FUNCTION_BLOCK AOI_StagingTemplate
VAR_INPUT
	execute : BOOL;
END_VAR
VAR_IN_OUT
	materialsArr : ARRAY[*] OF PositionMaterials; //[0..GVL.maxPairs]
	table : StagingTable;
END_VAR
VAR_INPUT
	includeTop, includeLeft, includeRight, includeBottom : BOOL; 
END_VAR
VAR_OUTPUT
	busy : BOOL;
	done : BOOL;
END_VAR
VAR
	trigger : R_TRIG;
	run : BOOL;
	step : (IDLE, GENERATE, COMPLETE);
	i : INT;
END_VAR
VAR	
	stagingArray : ARRAY[0..(GVL.maxPairs+1)*2] OF STRING;
	
	template : StagingTable;
	templateSlots AT %M* : ARRAY[1..10] OF MaterialSlot;
END_VAR

{warning disable C0371}

template(slots:= templateSlots);

trigger(CLK:= execute, Q=> run);

CASE step OF
	IDLE:
		IF run THEN
			step := GENERATE;
			done := FALSE;
		END_IF
		
	GENERATE:
		//strings contain garbage chars after a null byte, they must be manually cleaned before checking if they are byte-empty
		CleanStringsArray(arr := stagingArray);
		IF ArrayIsEmpty(arr := ADR(stagingArray), arrSize := SIZEOF(stagingArray)) THEN //if staging array is empty, fill the array
			createStagingArray(
				includeTop:= includeTop, 
				includeLeft:= includeLeft, 
				includeRight:= includeRight, 
				includeBottom:= includeBottom);
		END_IF
		
		//copy over the real slots before autofilling, otherwise the template may fill occupied slots
		table.copyFrom(src := table);
		
		(*
		iterate through all pairs and autofill the template
		replace succesfully autofilled materials with empty string
		if staging needs to be performed a 2nd time, autofilling empty strings is always unsuccessful
		*)
		FOR i:=0 TO (GVL.maxPairs+1)*2 BY 1 DO
			IF template.autofill(material := stagingArray[i]) THEN
				stagingArray[i] := '';
			END_IF
		END_FOR
		
		step := COMPLETE;
	
	COMPLETE:
		done := TRUE;
		
		step := IDLE;
		
END_CASE

busy := run OR step > 0;

METHOD PRIVATE addToStagingArray : BOOL
VAR_INPUT
	material : STRING;
END_VAR
VAR
	remainingMaterial : STRING;
	splitMaterial : STRING;
END_VAR
remainingMaterial := material;
WHILE FIND(remainingMaterial, '_') > 0 DO
	splitCombinedMaterials(remainingMaterial, splitMaterial);
	IF splitMaterial <> '' THEN
		AddToStringArray(arr := stagingArray, newString := splitMaterial, numElements => , nextIndex => );
		(*
		AddToArray(
			arr := ADR(stagingArray), 
			numEntries := SIZEOF(stagingArray)/SIZEOF(stagingArray[0]), 
			dataSize := SIZEOF(STRING), 
			newEntry := splitMaterial);
		*)
	END_IF
END_WHILE

IF remainingMaterial <> '' THEN
	AddToStringArray(arr := stagingArray, newString := remainingMaterial, numElements => , nextIndex => );
	(*
	AddToArray(
		arr := ADR(stagingArray), 
		numEntries := SIZEOF(stagingArray)/SIZEOF(stagingArray[0]), 
		dataSize := SIZEOF(STRING), 
		newEntry := remainingMaterial);
	*)
END_IF

addToStagingArray := TRUE;
END_METHOD

METHOD clearArray : BOOL
VAR_INPUT
END_VAR
MEMSET(ADR(stagingArray), 0, SIZEOF(stagingArray));
END_METHOD

METHOD clearTemplate : BOOL
VAR_INPUT
END_VAR
template.clear();
END_METHOD

METHOD PRIVATE createStagingArray : BOOL
VAR_INPUT
	includeTop : BOOL;
	includeLeft : BOOL;
	includeRight : BOOL;
	includeBottom : BOOL;
END_VAR
VAR
	remainingMaterial : STRING;
	splitMaterial : STRING;
	
	i : INT;
END_VAR
FOR i:=0 TO GVL.maxPairs BY 1 DO
	IF includeTop THEN
		addToStagingArray(material := materialsArr[i].top);
	END_IF
	
	IF includeLeft THEN
		addToStagingArray(material := materialsArr[i].left);
	END_IF
	
	IF includeRight THEN
		addToStagingArray(material := materialsArr[i].right);
	END_IF
	
	IF includeBottom THEN
		addToStagingArray(material := materialsArr[i].bottom);
	END_IF
END_FOR
END_METHOD

METHOD getSlot : STRING
VAR_INPUT
	i : INT;
END_VAR
VAR_OUTPUT
	error : BOOL;
END_VAR
getSlot := template.getSlot(i := i, error => error);
END_METHOD

METHOD reset : BOOL
VAR_INPUT
END_VAR
VAR
	temp : AOI_StagingTemplate;
END_VAR
//(*
busy := FALSE;
done := FALSE;
step := 0;

clearArray();
clearTemplate();
//*)
//THIS^ := temp;
END_METHOD

METHOD PRIVATE splitCombinedMaterials : BOOL
VAR_IN_OUT
	materialID : STRING;
	splitMaterial : STRING;
END_VAR
VAR
	i : INT;
END_VAR
FindAndSplitChar(
	sSeparatorChar:= '_', 
	pSrcString:= ADR(materialID), 
	
	pLeftString:= ADR(splitMaterial), 
	nLeftSize:= SIZEOF(splitMaterial), 
	
	pRightString:= ADR(materialID), 
	nRightSize:= SIZEOF(materialID), 
	
	bSearchFromRight:= FALSE);
END_METHOD

END_FUNCTION_BLOCK

(* stored: Version 1.1.0.1, ProductVersion 3.1.4024.11
   POU AOI_StagingTemplate: Id {0037dd5b-bbfe-4f9c-ade0-ad27a646a516}, SpecialFunc None
   Folder Private: Id {3c6bf1e6-e944-469b-bcd7-a97f56b268e0}
   Method addToStagingArray: Id {655ab137-48d6-43ef-8a47-92e88a7eb6e3}
   Method clearArray: Id {c4d9cbd8-5b02-4798-84d6-92f71b58ca65}
   Method clearTemplate: Id {0b1de681-f998-4280-8661-36d9e7be5728}
   Method createStagingArray: Id {e33729e2-b40e-4f85-bcc3-df064c30aeb0}
   Method getSlot: Id {20858403-7499-4509-b232-807eaa0bca7e}
   Method reset: Id {30967273-5971-4694-a3f9-4830fbeea9d0}
   Method splitCombinedMaterials: Id {419e2fad-7d72-4697-81cf-ab6b3eae18e9} *)
